% RSLogix 500 project P6 - Hourmeter.RSS, saved by version 8.30.00.16 %
PROJECT "P6"    % processor: Bul.1763 MicroLogix 1100 Series B %

PROGRAM FILES
  LAD 2 "MAIN"  3 rungs
  LAD 3 "IO"  2 rungs
  LAD 4 "LOGIC"  6 rungs

DATA FILES
  O0 OUTPUT  4 elements
  I1 INPUT  6 elements
  S2 STATUS  66 elements
  B3 BINARY  1 elements
  T4 TIMER  1 elements
  C5 COUNTER  3 elements
  R6 CONTROL  1 elements
  N7 INTEGER  4 elements
  F8 FLOAT  1 elements

LADDER 2 "MAIN"
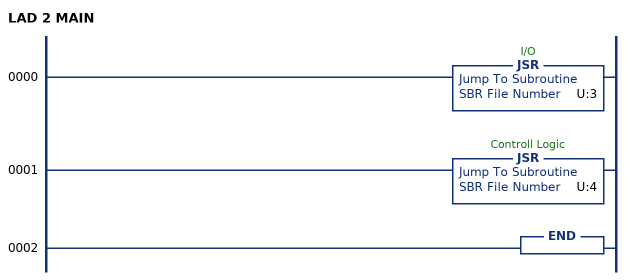
% Rung: 0 %
SOR JSR U:3 EOR
%   U:3  "I/O" %
% Rung: 1 %
SOR JSR U:4 EOR
%   U:4  "Controll Logic" %
% Rung: 2 %
SOR END EOR

LADDER 3 "IO"
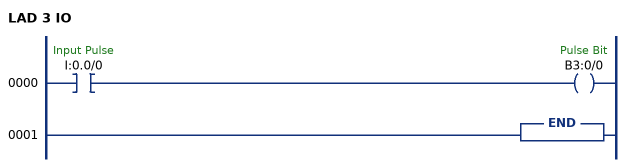
% Rung: 0 %
SOR XIC I:0.0/0 OTE B3:0/0 EOR
%   I:0.0/0  "Input Pulse" %
%   B3:0/0  "Pulse Bit" %
% Rung: 1 %
SOR END EOR

LADDER 4 "LOGIC"
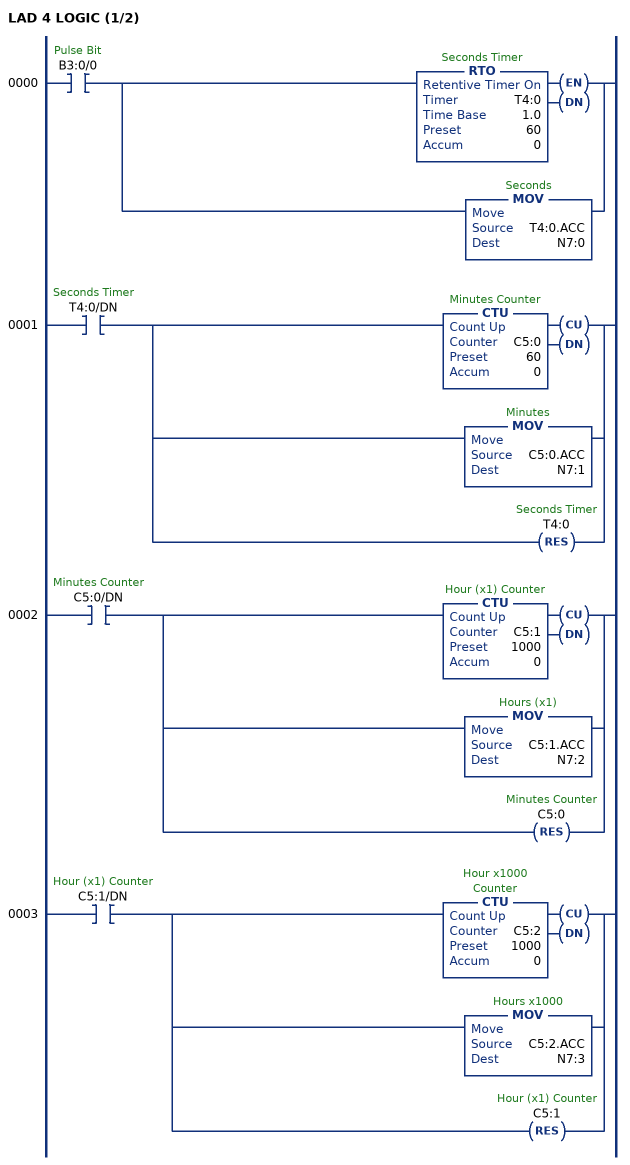
% Rung: 0 %
SOR XIC B3:0/0 BST RTO T4:0 1.0 60 0 NXB MOV T4:0.ACC N7:0 BND EOR
%   B3:0/0  "Pulse Bit" %
%   T4:0  "Seconds Timer" %
%   N7:0  "Seconds" %
% Rung: 1 %
SOR XIC T4:0/DN BST CTU C5:0 60 0 NXB MOV C5:0.ACC N7:1 NXB RES T4:0 BND EOR
%   T4:0  "Seconds Timer" %
%   C5:0  "Minutes Counter" %
%   N7:1  "Minutes" %
% Rung: 2 %
SOR XIC C5:0/DN BST CTU C5:1 1000 0 NXB MOV C5:1.ACC N7:2 NXB RES C5:0 BND EOR
%   C5:0  "Minutes Counter" %
%   C5:1  "Hour (x1) Counter" %
%   N7:2  "Hours (x1)" %
% Rung: 3 %
SOR XIC C5:1/DN BST CTU C5:2 1000 0 NXB MOV C5:2.ACC N7:3 NXB RES C5:1 BND EOR
%   C5:1  "Hour (x1) Counter" %
%   C5:2  "Hour x1000 Counter" %
%   N7:3  "Hours x1000" %

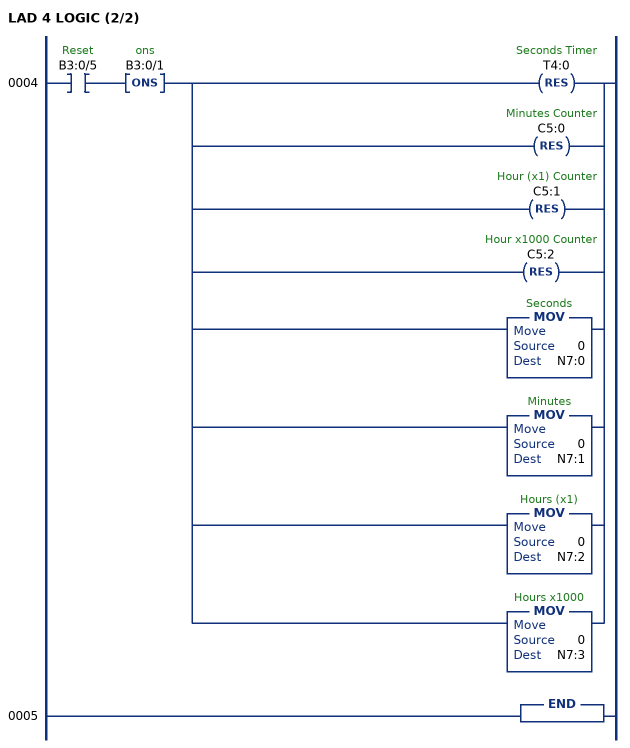
% Rung: 4 %
SOR XIC B3:0/5 ONS B3:0/1 BST RES T4:0 NXB RES C5:0 NXB RES C5:1 NXB RES C5:2 NXB MOV 0 N7:0 NXB MOV 0 N7:1 NXB MOV 0 N7:2 NXB MOV 0 N7:3 BND EOR
%   B3:0/5  "Reset" %
%   B3:0/1  "ons" %
%   T4:0  "Seconds Timer" %
%   C5:0  "Minutes Counter" %
%   C5:1  "Hour (x1) Counter" %
%   C5:2  "Hour x1000 Counter" %
%   N7:0  "Seconds" %
%   N7:1  "Minutes" %
%   N7:2  "Hours (x1)" %
%   N7:3  "Hours x1000" %
% Rung: 5 %
SOR END EOR

OTHER DOCUMENTED ADDRESSES
  B3:0/2  "ons"
  B3:0/3  "ons"
  B3:0/4  "ons"

DATA TABLE (non-zero values as saved)
DATA T4
% .PRE .ACC %
% T4:0 % 60 0
DATA C5
% .PRE .ACC %
% C5:0 % 60 0
% C5:1 % 1000 0
% C5:2 % 1000 0
